FUNCTION_BLOCK XtsMotorModule EXTENDS CyclicBase
VAR_INPUT
END_VAR
VAR_OUTPUT
END_VAR
VAR
END_VAR

METHOD PUBLIC  Cycle : HRESULT
VAR_INPUT
END_VAR
END_METHOD

METHOD Initialise : HRESULT
VAR_INPUT
END_VAR
END_METHOD

END_FUNCTION_BLOCK

(* stored: Version 1.1.0.1, ProductVersion 3.1.4024.12
   POU XtsMotorModule: Id {447db564-ab24-433c-b078-4cedd1c7411e}, SpecialFunc None
   Method Cycle: Id {1188f197-bbd0-4970-903a-af249f1ed9e0}
   Method Initialise: Id {0d230f78-299f-458d-bcac-a537a1290197} *)
